// TIA Portal V19 export
FUNCTION "ctrlIo" : Void   // FC2, LAD
{ S7_Optimized_Access := 'TRUE' }
// stored: SetENOAutomatically false
   VAR_INPUT
      input : Bool;
   END_VAR
   VAR_OUTPUT
      output : Bool;
   END_VAR
BEGIN

REGION Network 1
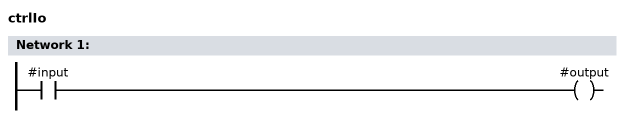
   RUNG wire#powerrail
      Contact( #input )
      Coil( #output )
   END_RUNG
   // the same network as SCL:
   #output := #input;
END_REGION
END_FUNCTION
